FUNCTION_BLOCK FILTER_MAV_W_Test EXTENDS FB_TestSuite
VAR_INPUT
END_VAR
VAR_OUTPUT
END_VAR
VAR
END_VAR

AverageEightThenTenEqualsNine();
AverageTenThenEightEqualsNine();

METHOD AverageEightThenTenEqualsNine
VAR
	MAV : FILTER_MAV_W;
	Result : WORD;
	ExpectedAverage : WORD := 9;
END_VAR
TEST('AverageEightThenTenEqualsNine');
 
MAV(X := 8, N := 2);
MAV(X := 10, Y => Result);
 
AssertEquals(Expected := ExpectedAverage,
             Actual := Result,
             Message := 'The calculation is not correct');
 
TEST_FINISHED();
END_METHOD

METHOD AverageTenThenEightEqualsNine
VAR
	MAV : FILTER_MAV_W;
	Result : WORD;
	ExpectedAverage : WORD := 9;
END_VAR
TEST('AverageTenThenEightEqualsNine');
 
MAV(X := 10, N := 2);
MAV(X := 8, Y => Result);
 
AssertEquals(Expected := ExpectedAverage,
             Actual := Result,
             Message := 'The calculation is not correct');
 
TEST_FINISHED();
END_METHOD

END_FUNCTION_BLOCK

(* stored: Version 1.1.0.1, ProductVersion 3.1.4024.9
   POU FILTER_MAV_W_Test: Id {6afb04ac-795a-4ebe-b33c-51570d47894d}, SpecialFunc None
   Method AverageEightThenTenEqualsNine: Id {85965441-dcfa-4ab0-9560-2d610c5e3a73}
   Method AverageTenThenEightEqualsNine: Id {116ad14c-174a-4dd4-a9a6-807c4fe2ecac} *)
